TYPE ST_CalibrationData :
STRUCT
	dDateTime 		: STRING(32);
	iPumpNumber 	: USINT;
	sStep			: STRING(64);
	rTareWeigth		: LREAL;
	rGrossWeigth 	: LREAL;
	rNetWeigth		: LREAL;
	rNetVolume		: LREAL;
	rTargetVolume	: LREAL;
	rDifferencePercent	: LREAL;
	rDifferenceUl	: LREAL;
	rCriteria		: REAL;
	iPumpRevs		: UINT;
END_STRUCT
END_TYPE

(* stored: Version 1.1.0.1, ProductVersion 3.1.4024.12
   DUT ST_CalibrationData: Id {afee19e0-65bb-42e5-a931-500e7dce160f} *)
